{attribute addProperty BoxType "EJ5151-0000-0016"}
{attribute addProperty Id "Period_valueAT %I*UDINT324"}
{attribute addProperty CRC "2891036832"}
{attribute addProperty SizeInBites "32"}
{attribute addProperty SizeInBytes "4"}
TYPE ENC_Inputs_AC51B8A0 :
STRUCT
	{attribute addProperty Name "Period_value"}
	Period_value AT %I* : UDINT;
END_STRUCT
END_TYPE

(* stored: Version 1.2.0.0, ProductVersion 3.1.4024.9
   DUT ENC_Inputs_AC51B8A0: Id {38e09eb8-ad41-432a-b5d5-bbf348af66aa} *)
